TYPE TcaEngelCastingCarrierJob :
STRUCT
	RequestNoCarrier : BOOL;	// TRUE wenn kein neuer Werkstückträger benötigt wird -> Ablage wird leer gemacht
	RequestCarrier : BOOL;		// TRUE wenn ein neuer Werkstückträger benötigt wird
	CarrierId : INT;			// ID vom Werkstückträger, Geometrischen Daten werden auf der Engel Steuerung verwaltet
	Empty : BOOL;				// TRUE wenn ein Werkstückträger mir leeren Plätzen benötigt wird
	Unfinished : BOOL;			// TRUE wenn ein Werkstückträger mit unfertigen Werkstücken benötigt wird
END_STRUCT
END_TYPE

(* stored: Version 1.1.0.1
   DUT TcaEngelCastingCarrierJob: Id {3fe88b83-8e07-4c94-bf8e-b68599957a3a} *)
